Universal Robots PolyScope program: Aufgabe1_1.urp

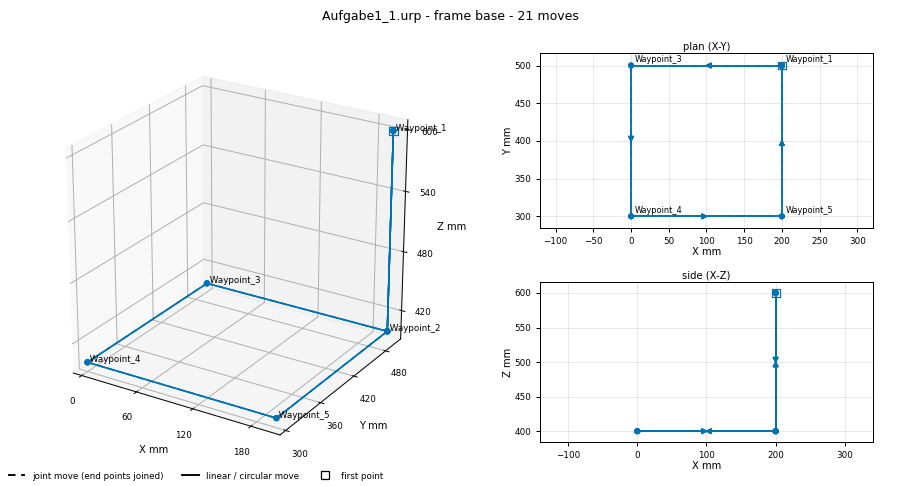
[picture p0: tool path of Aufgabe1_1.urp in frame base, 21 of 21 moves have a stored position in this frame; points joined in program order, loops and branches not executed]
Program Aufgabe1_1 (installation=Aufgabe1_1 directory=/home/ur/ursim-current/programs/new folder_1 createdIn=5.12.4.1101661 lastSavedIn=5.12.4.1101661 robotSerialNumber=20195299999)
Calibrated DH parameters: a=[0, -0.6127, -0.57155, 0, 0, 0]; d=[0.1807, 0, 0, 0.17415, 0.11985, 0.11655]; alpha=[1.570796, 0, 0, 1.570796, -1.570796, 0]; deltaTheta=[0, 0, 0, 0, 0, 0]
Robot Program (runOnlyOnce=false)
  MoveJ speed 60 deg/s, acceleration 80 deg/s^2 (useActiveTCP=true) feature=Base
    Waypoint Waypoint_1: TCP in base x=200 y=500 z=600 mm, rx=0 ry=3.1416 rz=0 rad; joints [-130.669, -107.049, -247.94, -95.011, -90, -220.669] deg
    MoveJ speed 60 deg/s, acceleration 80 deg/s^2 (useActiveTCP=true) feature=Base
      Waypoint Waypoint_2: TCP in base x=200 y=500 z=400 mm, rx=0 ry=3.1416 rz=0 rad; joints [-130.669, -100.942, -231.354, -117.703, -90, -220.669] deg
      Waypoint Waypoint_3: TCP in base x=0 y=500 z=400 mm, rx=0 ry=3.1416 rz=0 rad; joints [-110.383, -105.404, -228.116, -116.479, -90, -200.383] deg
      Waypoint Waypoint_4: TCP in base x=0 y=300 z=400 mm, rx=0 ry=3.1416 rz=0 rad; joints [-125.486, -135.885, -214.989, -99.126, -90, -215.486] deg
      Waypoint Waypoint_5: TCP in base x=200 y=300 z=400 mm, rx=0 ry=3.1416 rz=0 rad; joints [-152.572, -124.944, -218.131, -106.925, -90, -242.572] deg
      Waypoint Waypoint_2: TCP in base x=200 y=500 z=400 mm, rx=0 ry=3.1416 rz=0 rad; joints [-130.669, -100.942, -231.354, -117.703, -90, -220.669] deg
    MoveJ speed 60 deg/s, acceleration 80 deg/s^2 (useActiveTCP=true) feature=Base
      Waypoint Waypoint_1: TCP in base x=200 y=500 z=600 mm, rx=0 ry=3.1416 rz=0 rad; joints [-130.669, -107.049, -247.94, -95.011, -90, -220.669] deg
  MoveL speed 250 mm/s, acceleration 1200 mm/s^2 (useActiveTCP=true) feature=Base
    Waypoint Waypoint_1: TCP in base x=200 y=500 z=600 mm, rx=0 ry=3.1416 rz=0 rad; joints [-130.669, -107.049, -247.94, -95.011, -90, -220.669] deg
    MoveL speed 250 mm/s, acceleration 1200 mm/s^2 (useActiveTCP=true) feature=Base
      Waypoint Waypoint_2: TCP in base x=200 y=500 z=400 mm, rx=0 ry=3.1416 rz=0 rad; joints [-130.669, -100.942, -231.354, -117.703, -90, -220.669] deg
      Waypoint Waypoint_3: TCP in base x=0 y=500 z=400 mm, rx=0 ry=3.1416 rz=0 rad; joints [-110.383, -105.404, -228.116, -116.479, -90, -200.383] deg
      Waypoint Waypoint_4: TCP in base x=0 y=300 z=400 mm, rx=0 ry=3.1416 rz=0 rad; joints [-125.486, -135.885, -214.989, -99.126, -90, -215.486] deg
      Waypoint Waypoint_5: TCP in base x=200 y=300 z=400 mm, rx=0 ry=3.1416 rz=0 rad; joints [-152.572, -124.944, -218.131, -106.925, -90, -242.572] deg
      Waypoint Waypoint_2: TCP in base x=200 y=500 z=400 mm, rx=0 ry=3.1416 rz=0 rad; joints [-130.669, -100.942, -231.354, -117.703, -90, -220.669] deg
    MoveL speed 250 mm/s, acceleration 1200 mm/s^2 (useActiveTCP=true) feature=Base
      Waypoint Waypoint_1: TCP in base x=200 y=500 z=600 mm, rx=0 ry=3.1416 rz=0 rad; joints [-130.669, -107.049, -247.94, -95.011, -90, -220.669] deg
  MoveP speed 250 mm/s, acceleration 1200 mm/s^2 (blendRadius=0.025 useActiveTCP=true) feature=Base
    Waypoint Waypoint_1: TCP in base x=200 y=500 z=600 mm, rx=0 ry=3.1416 rz=0 rad; joints [-130.669, -107.049, -247.94, -95.011, -90, -220.669] deg
    MoveP speed 250 mm/s, acceleration 1200 mm/s^2 (blendRadius=0.025 useActiveTCP=true) feature=Base
      Waypoint Waypoint_2: TCP in base x=200 y=500 z=400 mm, rx=0 ry=3.1416 rz=0 rad; joints [-130.669, -100.942, -231.354, -117.703, -90, -220.669] deg
      Waypoint Waypoint_3: TCP in base x=0 y=500 z=400 mm, rx=0 ry=3.1416 rz=0 rad; joints [-110.383, -105.404, -228.116, -116.479, -90, -200.383] deg
      Waypoint Waypoint_4: TCP in base x=0 y=300 z=400 mm, rx=0 ry=3.1416 rz=0 rad; joints [-125.486, -135.885, -214.989, -99.126, -90, -215.486] deg
      Waypoint Waypoint_5: TCP in base x=200 y=300 z=400 mm, rx=0 ry=3.1416 rz=0 rad; joints [-152.572, -124.944, -218.131, -106.925, -90, -242.572] deg
      Waypoint Waypoint_2: TCP in base x=200 y=500 z=400 mm, rx=0 ry=3.1416 rz=0 rad; joints [-130.669, -100.942, -231.354, -117.703, -90, -220.669] deg
    MoveP speed 250 mm/s, acceleration 1200 mm/s^2 (blendRadius=0.025 useActiveTCP=true) feature=Base
      Waypoint Waypoint_1: TCP in base x=200 y=500 z=600 mm, rx=0 ry=3.1416 rz=0 rad; joints [-130.669, -107.049, -247.94, -95.011, -90, -220.669] deg
